{attribute 'qualified_only'}
VAR_GLOBAL PERSISTENT
	testIncr :INT;
	testStr : SafeState;
	

END_VAR

(* stored: Version 1.1.0.1, ProductVersion 3.1.4022.12
   GVL GVL_Persistent: Id {045d5161-bee0-4560-be67-f10a5bc7eac4} *)
